INTERFACE I_AdsRW EXTENDS I_Component, I_TaskResult

{attribute 'monitoring' := 'call'}
PROPERTY AmsNetId : T_AmsNetId
GET
END_GET
SET
END_SET
END_PROPERTY

{attribute 'monitoring' := 'call'}
PROPERTY AmsPort : T_AmsPort
GET
END_GET
SET
END_SET
END_PROPERTY

METHOD Read
VAR_INPUT
	IdxGrp	  : UDINT;
	IdxOffset : UDINT;
	pDestAddr : PVOID;
	Length	  : UDINT;
END_VAR
END_METHOD

METHOD ReadBySymbol
VAR_INPUT
	SymbolName : STRING(255);
	pDestAddr  : PVOID;
	Length	   : UDINT;
END_VAR
END_METHOD

METHOD Write
VAR_INPUT
	IdxGrp		: UDINT;
	IdxOffset	: UDINT;
	pSourceAddr : PVOID;
	Length		: UDINT;
END_VAR
END_METHOD

METHOD WriteBySymbol
VAR_INPUT
	SymbolName	: STRING(255);
	pSourceAddr : PVOID;
	Length		: UDINT;
END_VAR
END_METHOD

END_INTERFACE

(* stored: Version 1.1.0.1, ProductVersion 3.1.4026.18
   Itf I_AdsRW: Id {d9aa18d4-eb01-40f5-a4f4-d7eed26c68d9}
   Property AmsNetId: Id {a31ac575-5849-4a93-879d-acde219d0a22}
   Get Get: Id {89cdff9c-c6c0-4ebb-91df-37712933f442}
   Set Set: Id {c319ab37-9ecb-48ad-904e-983bc99bc235}
   Property AmsPort: Id {85438c3a-36ce-4644-92a2-db52ba7c989c}
   Get Get: Id {115c8295-2ed1-4bd5-96fc-f4b15f03e523}
   Set Set: Id {da8cba4a-5d64-47a4-83ae-28bb7ff46c2e}
   Method Read: Id {9d80728c-85ea-4c1d-8679-9e32b12b4701}
   Method ReadBySymbol: Id {0c44b531-128e-4416-b728-cec20b5a69cc}
   Method Write: Id {153567fa-e59c-404d-a88c-d2b7c15415b1}
   Method WriteBySymbol: Id {741e5885-8959-436f-9225-620933a482e4} *)
